TYPE E_TriggerOutput :
(
	PlcOutput,
	TripleTriggerModul,
	MultiZOutput,
	MultiZPWM
)USINT;
END_TYPE

(* stored: Version 1.1.0.1, ProductVersion 3.1.4024.6
   DUT E_TriggerOutput: Id {38ee990a-2463-4494-b256-da57c2c52737} *)
